// TIA Portal V18 export
DATA_BLOCK "ER_SIREN_ON_WNER_count_change"   // DB41
VERSION : 0.1
// stored: AutoNumber true, DBAccessibleFromOPCUA true, InstanceOfName I_TRIG_int_change, InstanceOfType FB
"I_TRIG_int_change"
   // VAR_INPUT
   //    J : Int;
   // END_VAR
   // VAR_OUTPUT
   //    C : Bool;
   // END_VAR
   // VAR
   //    J_was : Int;
   // END_VAR
BEGIN
END_DATA_BLOCK
